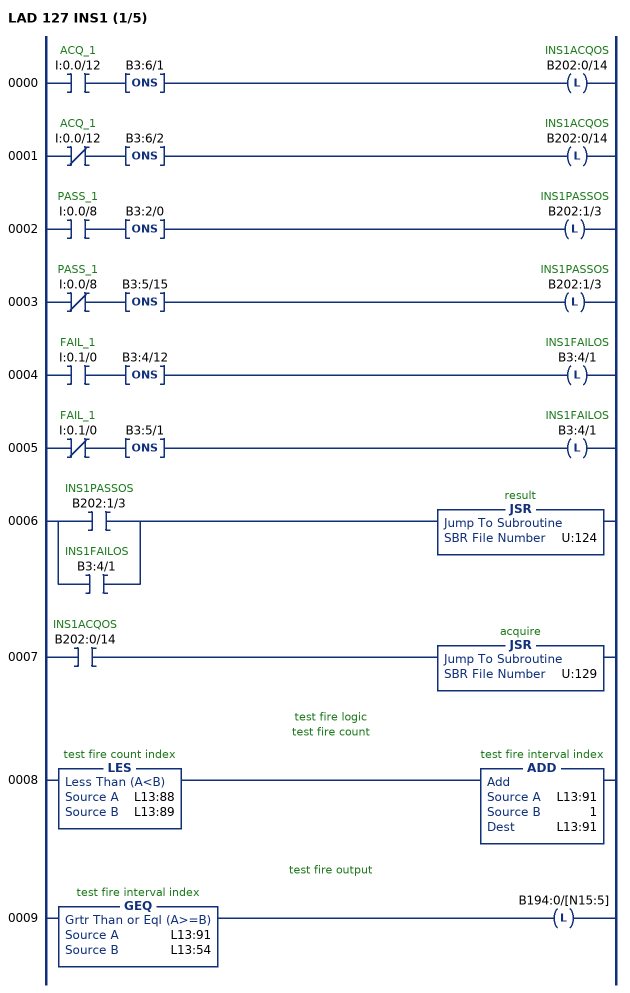
% Rung: 0 %
SOR XIC I:0.0/12 ONS B3:6/1 OTL B202:0/14 EOR
%   I:0.0/12  ACQ_1 %
%   B202:0/14  INS1ACQOS %
% Rung: 1 %
SOR XIO I:0.0/12 ONS B3:6/2 OTL B202:0/14 EOR
%   I:0.0/12  ACQ_1 %
%   B202:0/14  INS1ACQOS %
% Rung: 2 %
SOR XIC I:0.0/8 ONS B3:2/0 OTL B202:1/3 EOR
%   I:0.0/8  PASS_1 %
%   B202:1/3  INS1PASSOS %
% Rung: 3 %
SOR XIO I:0.0/8 ONS B3:5/15 OTL B202:1/3 EOR
%   I:0.0/8  PASS_1 %
%   B202:1/3  INS1PASSOS %
% Rung: 4 %
SOR XIC I:0.1/0 ONS B3:4/12 OTL B3:4/1 EOR
%   I:0.1/0  FAIL_1 %
%   B3:4/1  INS1FAILOS %
% Rung: 5 %
SOR XIO I:0.1/0 ONS B3:5/1 OTL B3:4/1 EOR
%   I:0.1/0  FAIL_1 %
%   B3:4/1  INS1FAILOS %
% Rung: 6 %
SOR BST XIC B202:1/3 NXB XIC B3:4/1 BND JSR U:124 EOR
%   B202:1/3  INS1PASSOS %
%   B3:4/1  INS1FAILOS %
%   U:124  "result" %
% Rung: 7 %
SOR XIC B202:0/14 JSR U:129 EOR
%   B202:0/14  INS1ACQOS %
%   U:129  "acquire" %
% Rung: 8 %
% test fire logic
% 
% test fire count %
SOR LES L13:88 L13:89 ADD L13:91 1 L13:91 EOR
%   L13:88  "test fire count index" %
%   L13:89  "test fire count" %
%   L13:91  "test fire interval index" %
% Rung: 9 %
% test fire output %
SOR GEQ L13:91 L13:54 OTL B194:0/[N15:5] EOR
%   L13:91  "test fire interval index" %
%   L13:54  "test fire interval" %
%   N15:5  INS_1_TRIG_LOC %

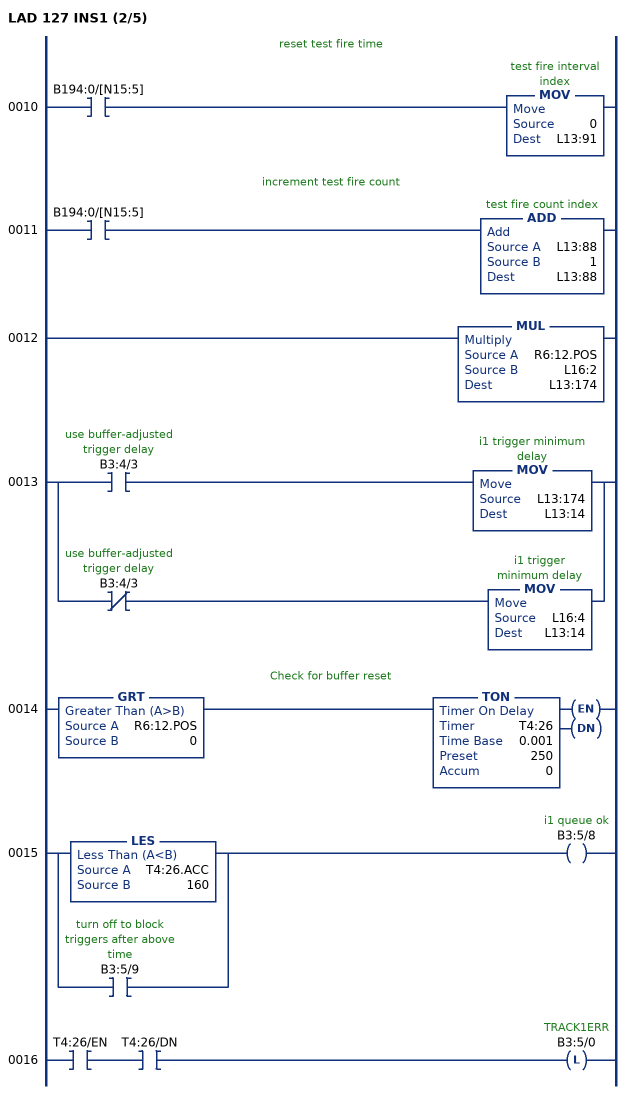
% Rung: 10 %
% reset test fire time %
SOR XIC B194:0/[N15:5] MOV 0 L13:91 EOR
%   N15:5  INS_1_TRIG_LOC %
%   L13:91  "test fire interval index" %
% Rung: 11 %
% increment test fire count %
SOR XIC B194:0/[N15:5] ADD L13:88 1 L13:88 EOR
%   N15:5  INS_1_TRIG_LOC %
%   L13:88  "test fire count index" %
% Rung: 12 %
SOR MUL R6:12.POS L16:2 L13:174 EOR
%   L16:2  TRIG_DELAY_Q_MULTI %
% Rung: 13 %
SOR BST XIC B3:4/3 MOV L13:174 L13:14 NXB XIO B3:4/3 MOV L16:4 L13:14 BND EOR
%   B3:4/3  "use buffer-adjusted trigger delay" %
%   L13:14  "i1 trigger minimum delay" %
%   L16:4  TRIG_DELAY_FLAT_RATE %
% Rung: 14 %
% Check for buffer reset %
SOR GRT R6:12.POS 0 TON T4:26 0.001 250 0 EOR
% Rung: 15 %
SOR BST LES T4:26.ACC 160 NXB XIC B3:5/9 BND OTE B3:5/8 EOR
%   B3:5/9  "turn off to block triggers after above time" %
%   B3:5/8  "i1 queue ok" %
% Rung: 16 %
SOR XIC T4:26/EN XIC T4:26/DN OTL B3:5/0 EOR
%   B3:5/0  TRACK1ERR %

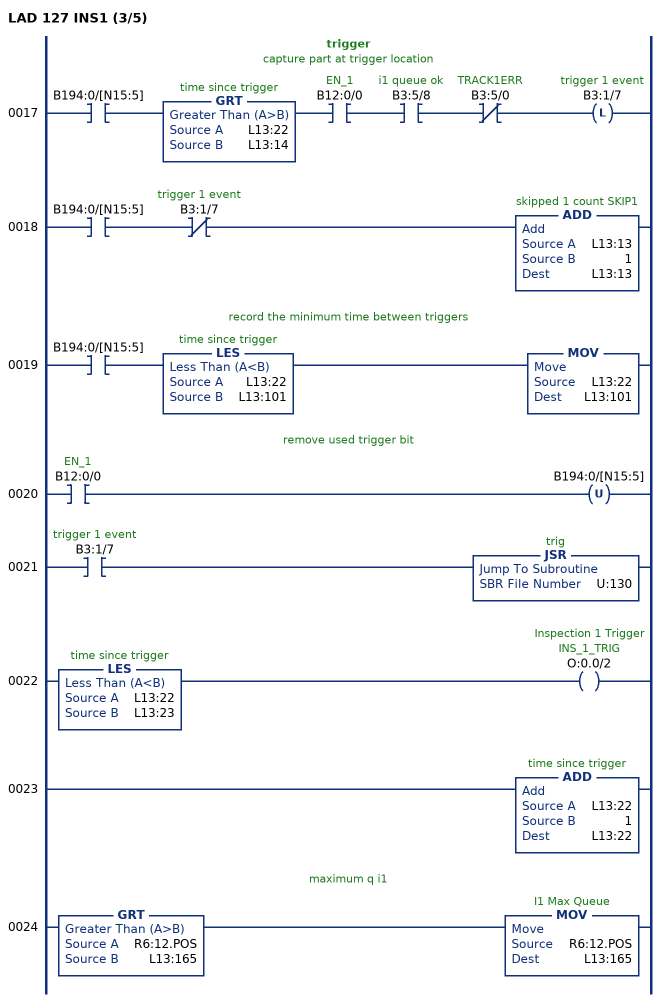
% Rung: 17 %
% TITLE: trigger %
% capture part at trigger location %
SOR XIC B194:0/[N15:5] GRT L13:22 L13:14 XIC B12:0/0 XIC B3:5/8 XIO B3:5/0 OTL B3:1/7 EOR
%   N15:5  INS_1_TRIG_LOC %
%   L13:22  "time since trigger" %
%   L13:14  "i1 trigger minimum delay" %
%   B12:0/0  EN_1 %
%   B3:5/8  "i1 queue ok" %
%   B3:5/0  TRACK1ERR %
%   B3:1/7  "trigger 1 event" %
% Rung: 18 %
SOR XIC B194:0/[N15:5] XIO B3:1/7 ADD L13:13 1 L13:13 EOR
%   N15:5  INS_1_TRIG_LOC %
%   B3:1/7  "trigger 1 event" %
%   L13:13  SKIP1  "skipped 1 count" %
% Rung: 19 %
% record the minimum time between triggers %
SOR XIC B194:0/[N15:5] LES L13:22 L13:101 MOV L13:22 L13:101 EOR
%   N15:5  INS_1_TRIG_LOC %
%   L13:22  "time since trigger" %
% Rung: 20 %
% remove used trigger bit %
SOR XIC B12:0/0 OTU B194:0/[N15:5] EOR
%   B12:0/0  EN_1 %
%   N15:5  INS_1_TRIG_LOC %
% Rung: 21 %
SOR XIC B3:1/7 JSR U:130 EOR
%   B3:1/7  "trigger 1 event" %
%   U:130  "trig" %
% Rung: 22 %
SOR LES L13:22 L13:23 OTE O:0.0/2 EOR
%   L13:22  "time since trigger" %
%   L13:23  "trigger on time" %
%   O:0.0/2  INS_1_TRIG  "Inspection 1 Trigger" %
% Rung: 23 %
SOR ADD L13:22 1 L13:22 EOR
%   L13:22  "time since trigger" %
% Rung: 24 %
% maximum q i1 %
SOR GRT R6:12.POS L13:165 MOV R6:12.POS L13:165 EOR
%   L13:165  "I1 Max Queue" %

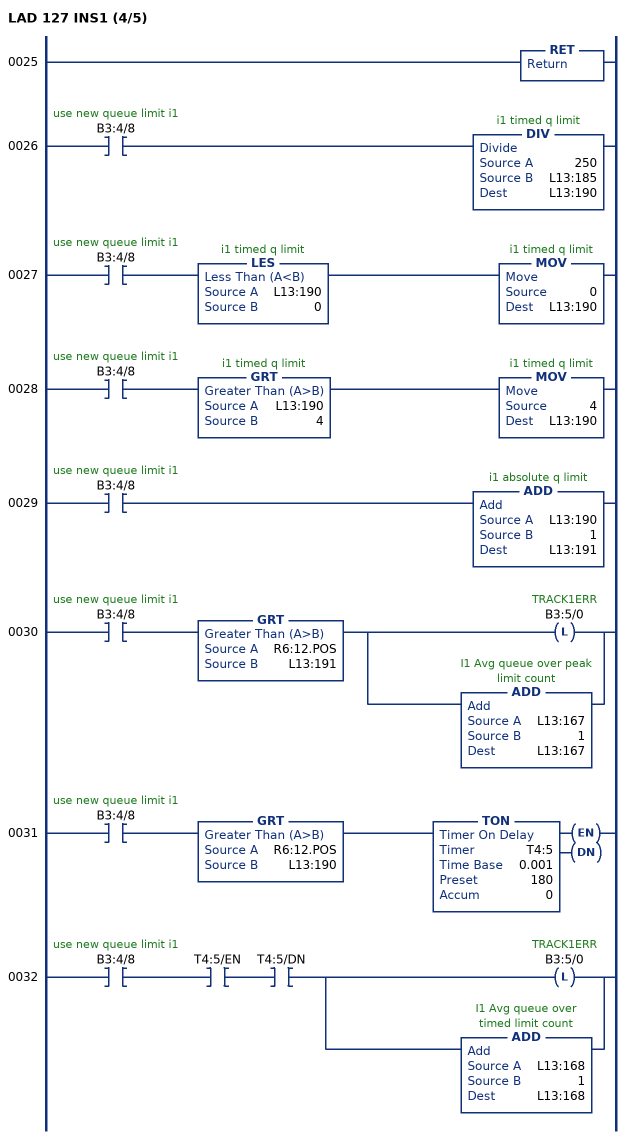
% Rung: 25 %
SOR RET EOR
% Rung: 26 %
SOR XIC B3:4/8 DIV 250 L13:185 L13:190 EOR
%   B3:4/8  "use new queue limit i1" %
%   L13:185  I1_TBT  "i1 average time between triggers" %
%   L13:190  "i1 timed q limit" %
% Rung: 27 %
SOR XIC B3:4/8 LES L13:190 0 MOV 0 L13:190 EOR
%   B3:4/8  "use new queue limit i1" %
%   L13:190  "i1 timed q limit" %
% Rung: 28 %
SOR XIC B3:4/8 GRT L13:190 4 MOV 4 L13:190 EOR
%   B3:4/8  "use new queue limit i1" %
%   L13:190  "i1 timed q limit" %
% Rung: 29 %
SOR XIC B3:4/8 ADD L13:190 1 L13:191 EOR
%   B3:4/8  "use new queue limit i1" %
%   L13:190  "i1 timed q limit" %
%   L13:191  "i1 absolute q limit" %
% Rung: 30 %
SOR XIC B3:4/8 GRT R6:12.POS L13:191 BST OTL B3:5/0 NXB ADD L13:167 1 L13:167 BND EOR
%   B3:4/8  "use new queue limit i1" %
%   L13:191  "i1 absolute q limit" %
%   B3:5/0  TRACK1ERR %
%   L13:167  "I1 Avg queue over peak limit count" %
% Rung: 31 %
SOR XIC B3:4/8 GRT R6:12.POS L13:190 TON T4:5 0.001 180 0 EOR
%   B3:4/8  "use new queue limit i1" %
%   L13:190  "i1 timed q limit" %
% Rung: 32 %
SOR XIC B3:4/8 XIC T4:5/EN XIC T4:5/DN BST OTL B3:5/0 NXB ADD L13:168 1 L13:168 BND EOR
%   B3:4/8  "use new queue limit i1" %
%   B3:5/0  TRACK1ERR %
%   L13:168  "I1 Avg queue over timed limit count" %

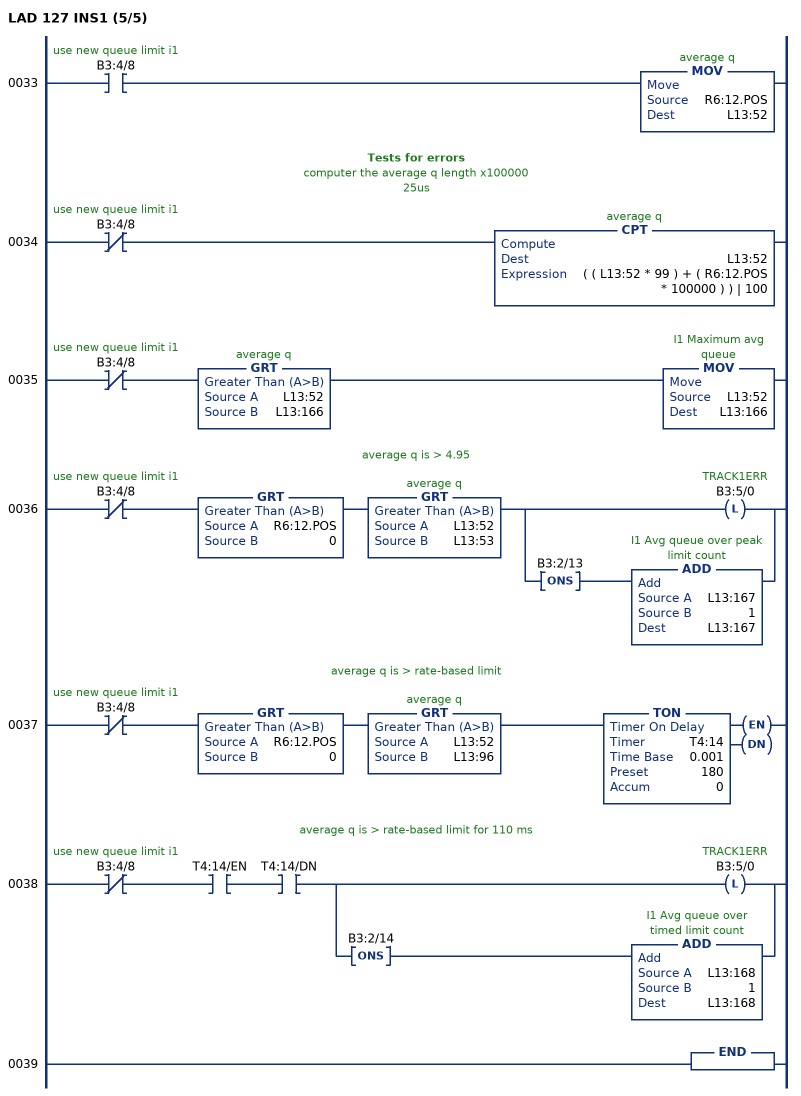
% Rung: 33 %
SOR XIC B3:4/8 MOV R6:12.POS L13:52 EOR
%   B3:4/8  "use new queue limit i1" %
%   L13:52  "average q" %
% Rung: 34 %
% TITLE: Tests for errors %
% computer the average q length x100000
% 25us %
SOR XIO B3:4/8 CPT L13:52 " ( ( L13:52 * 99 ) + ( R6:12.POS * 100000 ) ) | 100 " EOR
%   B3:4/8  "use new queue limit i1" %
%   L13:52  "average q" %
% Rung: 35 %
SOR XIO B3:4/8 GRT L13:52 L13:166 MOV L13:52 L13:166 EOR
%   B3:4/8  "use new queue limit i1" %
%   L13:52  "average q" %
%   L13:166  "I1 Maximum avg queue" %
% Rung: 36 %
% average q is > 4.95 %
SOR XIO B3:4/8 GRT R6:12.POS 0 GRT L13:52 L13:53 BST OTL B3:5/0 NXB ONS B3:2/13 ADD L13:167 1 L13:167 BND EOR
%   B3:4/8  "use new queue limit i1" %
%   L13:52  "average q" %
%   B3:5/0  TRACK1ERR %
%   L13:167  "I1 Avg queue over peak limit count" %
% Rung: 37 %
% average q is > rate-based limit %
SOR XIO B3:4/8 GRT R6:12.POS 0 GRT L13:52 L13:96 TON T4:14 0.001 180 0 EOR
%   B3:4/8  "use new queue limit i1" %
%   L13:52  "average q" %
%   L13:96  "i1 timed queue limit" %
% Rung: 38 %
% average q is > rate-based limit for 110 ms %
SOR XIO B3:4/8 XIC T4:14/EN XIC T4:14/DN BST OTL B3:5/0 NXB ONS B3:2/14 ADD L13:168 1 L13:168 BND EOR
%   B3:4/8  "use new queue limit i1" %
%   B3:5/0  TRACK1ERR %
%   L13:168  "I1 Avg queue over timed limit count" %
% Rung: 39 %
SOR END EOR

LADDER 128 "INS1PASS"
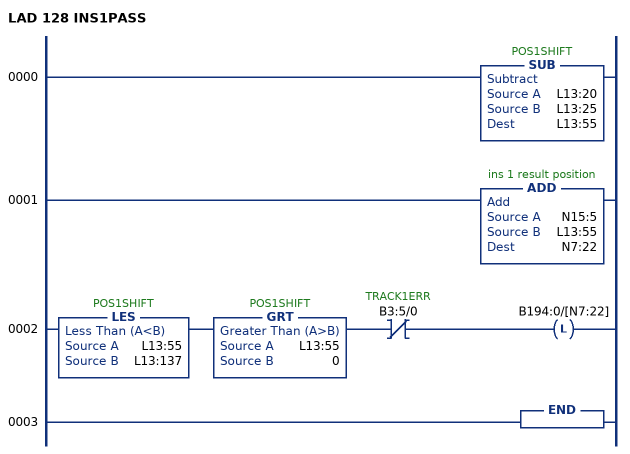
% Rung: 0 %
SOR SUB L13:20 L13:25 L13:55 EOR
%   L13:20  BOT_POSITION %
%   L13:25  POS1  "last acquisition position stamp" %
%   L13:55  POS1SHIFT %
% Rung: 1 %
SOR ADD N15:5 L13:55 N7:22 EOR
%   N15:5  INS_1_TRIG_LOC %
%   L13:55  POS1SHIFT %
%   N7:22  "ins 1 result position" %
% Rung: 2 %
SOR LES L13:55 L13:137 GRT L13:55 0 XIO B3:5/0 OTL B194:0/[N7:22] EOR
%   L13:55  POS1SHIFT %
%   B3:5/0  TRACK1ERR %
%   N7:22  "ins 1 result position" %
% Rung: 3 %
SOR END EOR

LADDER 129 "INS1ACQ"
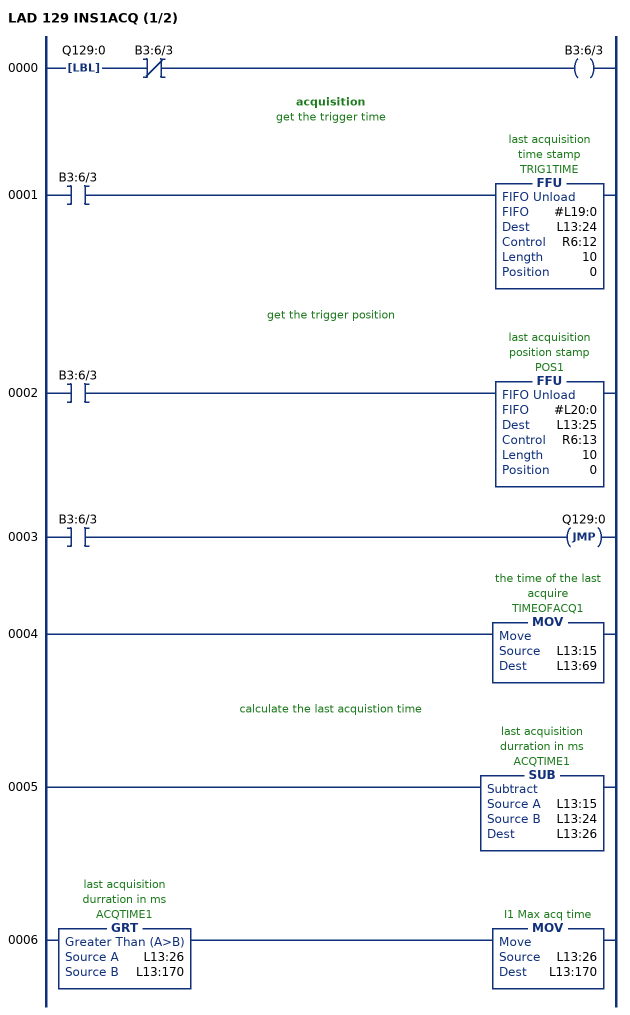
% Rung: 0 %
SOR LBL Q129:0 XIO B3:6/3 OTE B3:6/3 EOR
% Rung: 1 %
% TITLE: acquisition %
% get the trigger time %
SOR XIC B3:6/3 FFU #L19:0 L13:24 R6:12 10 0 EOR
%   L13:24  TRIG1TIME  "last acquisition time stamp" %
% Rung: 2 %
% get the trigger position %
SOR XIC B3:6/3 FFU #L20:0 L13:25 R6:13 10 0 EOR
%   L13:25  POS1  "last acquisition position stamp" %
% Rung: 3 %
SOR XIC B3:6/3 JMP Q129:0 EOR
% Rung: 4 %
SOR MOV L13:15 L13:69 EOR
%   L13:15  THE_TIME %
%   L13:69  TIMEOFACQ1  "the time of the last acquire" %
% Rung: 5 %
% calculate the last acquistion time %
SOR SUB L13:15 L13:24 L13:26 EOR
%   L13:15  THE_TIME %
%   L13:24  TRIG1TIME  "last acquisition time stamp" %
%   L13:26  ACQTIME1  "last acquisition durration in ms" %
% Rung: 6 %
SOR GRT L13:26 L13:170 MOV L13:26 L13:170 EOR
%   L13:26  ACQTIME1  "last acquisition durration in ms" %
%   L13:170  "I1 Max acq time" %

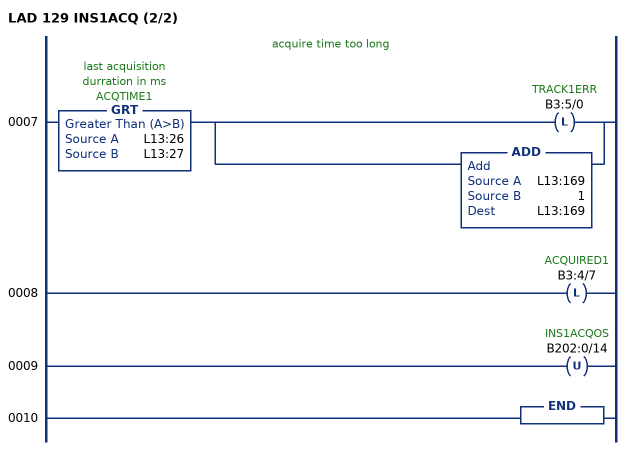
% Rung: 7 %
% acquire time too long %
SOR GRT L13:26 L13:27 BST OTL B3:5/0 NXB ADD L13:169 1 L13:169 BND EOR
%   L13:26  ACQTIME1  "last acquisition durration in ms" %
%   L13:27  "max acquisition time in ms" %
%   B3:5/0  TRACK1ERR %
% Rung: 8 %
SOR OTL B3:4/7 EOR
%   B3:4/7  ACQUIRED1 %
% Rung: 9 %
SOR OTU B202:0/14 EOR
%   B202:0/14  INS1ACQOS %
% Rung: 10 %
SOR END EOR

LADDER 130 "INS1TRIG"
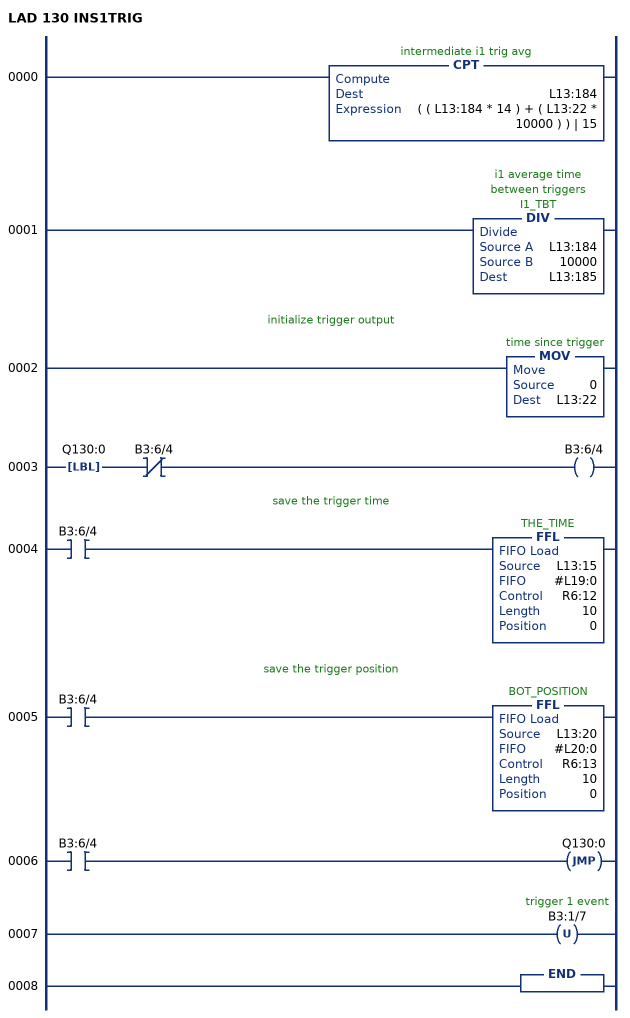
% Rung: 0 %
SOR CPT L13:184 " ( ( L13:184 * 14 ) + ( L13:22 * 10000 ) ) | 15 " EOR
%   L13:184  "intermediate i1 trig avg" %
%   L13:22  "time since trigger" %
% Rung: 1 %
SOR DIV L13:184 10000 L13:185 EOR
%   L13:184  "intermediate i1 trig avg" %
%   L13:185  I1_TBT  "i1 average time between triggers" %
% Rung: 2 %
% initialize trigger output %
SOR MOV 0 L13:22 EOR
%   L13:22  "time since trigger" %
% Rung: 3 %
SOR LBL Q130:0 XIO B3:6/4 OTE B3:6/4 EOR
% Rung: 4 %
% save the trigger time %
SOR XIC B3:6/4 FFL L13:15 #L19:0 R6:12 10 0 EOR
%   L13:15  THE_TIME %
% Rung: 5 %
% save the trigger position %
SOR XIC B3:6/4 FFL L13:20 #L20:0 R6:13 10 0 EOR
%   L13:20  BOT_POSITION %
% Rung: 6 %
SOR XIC B3:6/4 JMP Q130:0 EOR
% Rung: 7 %
SOR OTU B3:1/7 EOR
%   B3:1/7  "trigger 1 event" %
% Rung: 8 %
SOR END EOR

LADDER 131 "XFER"
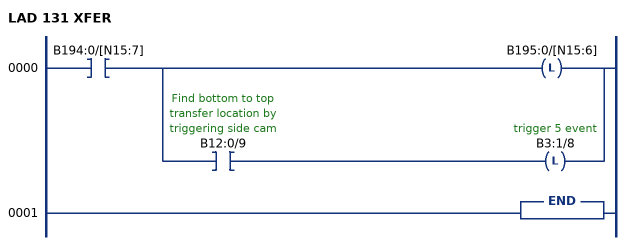
% Rung: 0 %
SOR XIC B194:0/[N15:7] BST OTL B195:0/[N15:6] NXB XIC B12:0/9 OTL B3:1/8 BND EOR
%   N15:7  XFER_OUT_LOC %
%   N15:6  XFER_IN_LOC %
%   B12:0/9  "Find bottom to top transfer location by triggering side cam" %
%   B3:1/8  "trigger 5 event" %
% Rung: 1 %
SOR END EOR

LADDER 140 "TOPOPTIC"
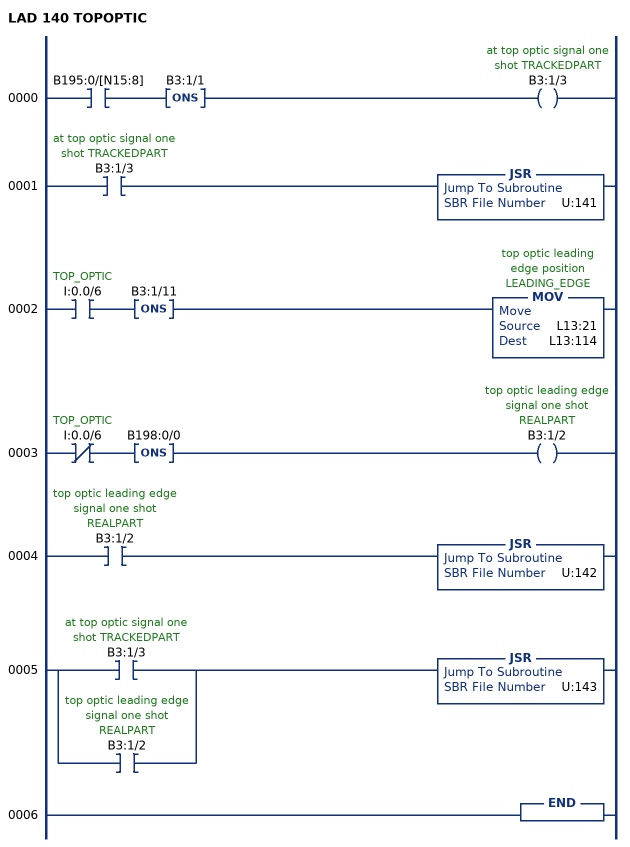
% Rung: 0 %
SOR XIC B195:0/[N15:8] ONS B3:1/1 OTE B3:1/3 EOR
%   N15:8  TOP_OPTIC_LOC %
%   B3:1/3  TRACKEDPART  "at top optic signal one shot" %
% Rung: 1 %
SOR XIC B3:1/3 JSR U:141 EOR
%   B3:1/3  TRACKEDPART  "at top optic signal one shot" %
% Rung: 2 %
SOR XIC I:0.0/6 ONS B3:1/11 MOV L13:21 L13:114 EOR
%   I:0.0/6  TOP_OPTIC %
%   L13:21  TOP_POSITION %
%   L13:114  LEADING_EDGE  "top optic leading edge position" %
% Rung: 3 %
SOR XIO I:0.0/6 ONS B198:0/0 OTE B3:1/2 EOR
%   I:0.0/6  TOP_OPTIC %
%   B3:1/2  REALPART  "top optic leading edge signal one shot" %
% Rung: 4 %
SOR XIC B3:1/2 JSR U:142 EOR
%   B3:1/2  REALPART  "top optic leading edge signal one shot" %
% Rung: 5 %
SOR BST XIC B3:1/3 NXB XIC B3:1/2 BND JSR U:143 EOR
%   B3:1/3  TRACKEDPART  "at top optic signal one shot" %
%   B3:1/2  REALPART  "top optic leading edge signal one shot" %
% Rung: 6 %
SOR END EOR

LADDER 141 "TOPOPVERT"
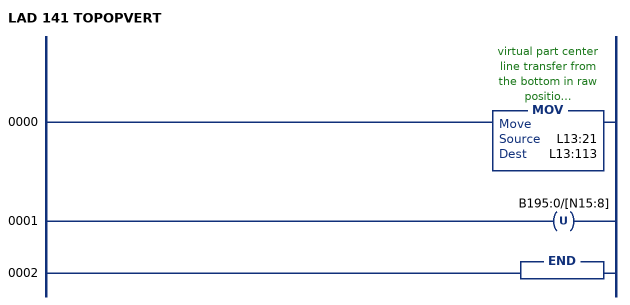
% Rung: 0 %
SOR MOV L13:21 L13:113 EOR
%   L13:21  TOP_POSITION %
%   L13:113  VERTUAL_PT_RAW_CL  "virtual part center line transfer from the bottom in raw position" %
% Rung: 1 %
SOR OTU B195:0/[N15:8] EOR
%   N15:8  TOP_OPTIC_LOC %
% Rung: 2 %
SOR END EOR

LADDER 142 "TOPOPREAL"
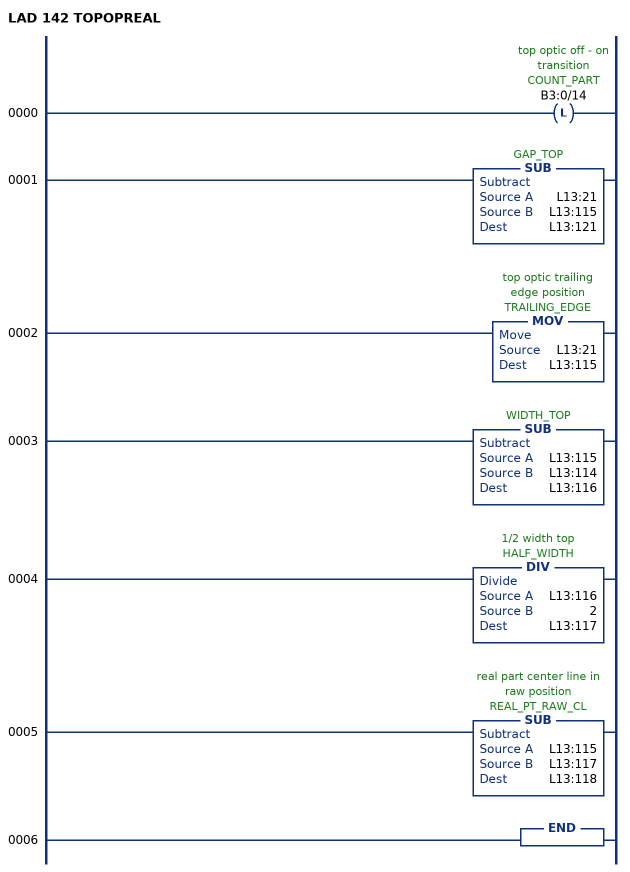
% Rung: 0 %
SOR OTL B3:0/14 EOR
%   B3:0/14  COUNT_PART  "top optic off - on transition" %
% Rung: 1 %
SOR SUB L13:21 L13:115 L13:121 EOR
%   L13:21  TOP_POSITION %
%   L13:115  TRAILING_EDGE  "top optic trailing edge position" %
%   L13:121  GAP_TOP %
% Rung: 2 %
SOR MOV L13:21 L13:115 EOR
%   L13:21  TOP_POSITION %
%   L13:115  TRAILING_EDGE  "top optic trailing edge position" %
% Rung: 3 %
SOR SUB L13:115 L13:114 L13:116 EOR
%   L13:115  TRAILING_EDGE  "top optic trailing edge position" %
%   L13:114  LEADING_EDGE  "top optic leading edge position" %
%   L13:116  WIDTH_TOP %
% Rung: 4 %
SOR DIV L13:116 2 L13:117 EOR
%   L13:116  WIDTH_TOP %
%   L13:117  HALF_WIDTH  "1/2 width top" %
% Rung: 5 %
SOR SUB L13:115 L13:117 L13:118 EOR
%   L13:115  TRAILING_EDGE  "top optic trailing edge position" %
%   L13:117  HALF_WIDTH  "1/2 width top" %
%   L13:118  REAL_PT_RAW_CL  "real part center line in raw position" %
% Rung: 6 %
SOR END EOR

LADDER 143 "TOPOPTEST"
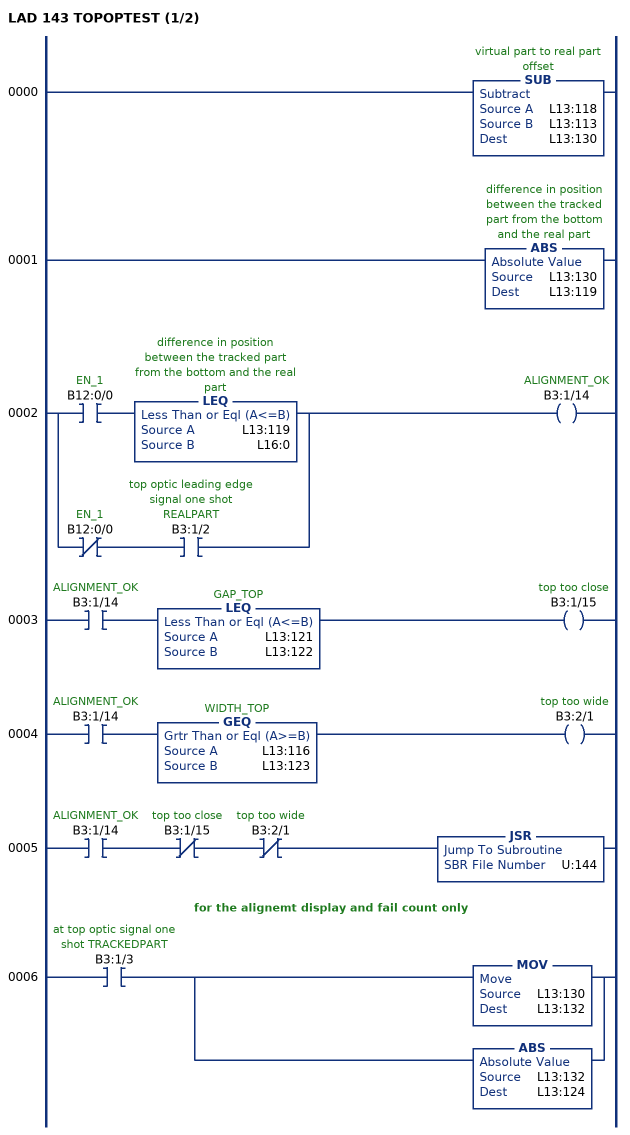
% Rung: 0 %
SOR SUB L13:118 L13:113 L13:130 EOR
%   L13:118  REAL_PT_RAW_CL  "real part center line in raw position" %
%   L13:113  VERTUAL_PT_RAW_CL  "virtual part center line transfer from the bottom in raw position" %
%   L13:130  "virtual part to real part offset" %
% Rung: 1 %
SOR ABS L13:130 L13:119 EOR
%   L13:130  "virtual part to real part offset" %
%   L13:119  "difference in position between the tracked part from the bottom and the real part" %
% Rung: 2 %
SOR BST XIC B12:0/0 LEQ L13:119 L16:0 NXB XIO B12:0/0 XIC B3:1/2 BND OTE B3:1/14 EOR
%   B12:0/0  EN_1 %
%   L13:119  "difference in position between the tracked part from the bottom and the real part" %
%   L16:0  MAX_OFFSET %
%   B3:1/2  REALPART  "top optic leading edge signal one shot" %
%   B3:1/14  ALIGNMENT_OK %
% Rung: 3 %
SOR XIC B3:1/14 LEQ L13:121 L13:122 OTE B3:1/15 EOR
%   B3:1/14  ALIGNMENT_OK %
%   L13:121  GAP_TOP %
%   L13:122  MIN_GAP_TOP %
%   B3:1/15  "top too close" %
% Rung: 4 %
SOR XIC B3:1/14 GEQ L13:116 L13:123 OTE B3:2/1 EOR
%   B3:1/14  ALIGNMENT_OK %
%   L13:116  WIDTH_TOP %
%   L13:123  MAX_WIDTH_TOP %
%   B3:2/1  "top too wide" %
% Rung: 5 %
SOR XIC B3:1/14 XIO B3:1/15 XIO B3:2/1 JSR U:144 EOR
%   B3:1/14  ALIGNMENT_OK %
%   B3:1/15  "top too close" %
%   B3:2/1  "top too wide" %
% Rung: 6 %
% TITLE: for the alignemt display and fail count only %
SOR XIC B3:1/3 BST MOV L13:130 L13:132 NXB ABS L13:132 L13:124 BND EOR
%   B3:1/3  TRACKEDPART  "at top optic signal one shot" %
%   L13:130  "virtual part to real part offset" %

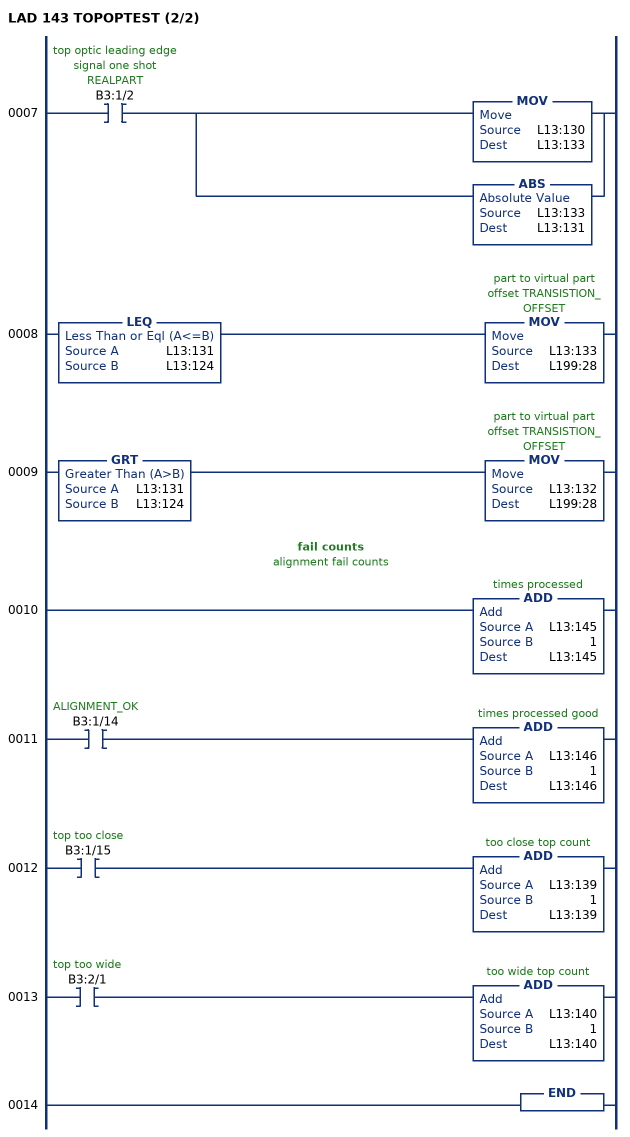
% Rung: 7 %
SOR XIC B3:1/2 BST MOV L13:130 L13:133 NXB ABS L13:133 L13:131 BND EOR
%   B3:1/2  REALPART  "top optic leading edge signal one shot" %
%   L13:130  "virtual part to real part offset" %
% Rung: 8 %
SOR LEQ L13:131 L13:124 MOV L13:133 L199:28 EOR
%   L199:28  TRANSISTION_OFFSET  "part to virtual part offset" %
% Rung: 9 %
SOR GRT L13:131 L13:124 MOV L13:132 L199:28 EOR
%   L199:28  TRANSISTION_OFFSET  "part to virtual part offset" %
% Rung: 10 %
% TITLE: fail counts %
% alignment fail counts %
SOR ADD L13:145 1 L13:145 EOR
%   L13:145  "times processed" %
% Rung: 11 %
SOR XIC B3:1/14 ADD L13:146 1 L13:146 EOR
%   B3:1/14  ALIGNMENT_OK %
%   L13:146  "times processed good" %
% Rung: 12 %
SOR XIC B3:1/15 ADD L13:139 1 L13:139 EOR
%   B3:1/15  "top too close" %
%   L13:139  "too close top count" %
% Rung: 13 %
SOR XIC B3:2/1 ADD L13:140 1 L13:140 EOR
%   B3:2/1  "top too wide" %
%   L13:140  "too wide top count" %
% Rung: 14 %
SOR END EOR

LADDER 144 "TOPOPOKAY"
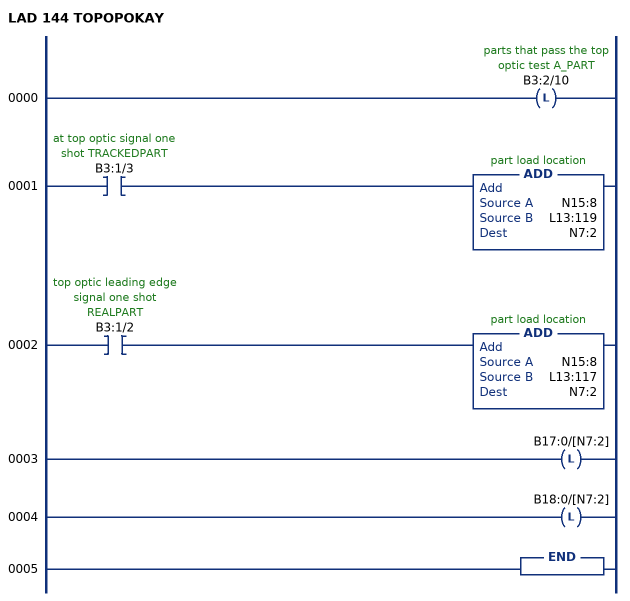
% Rung: 0 %
SOR OTL B3:2/10 EOR
%   B3:2/10  A_PART  "parts that pass the top optic test" %
% Rung: 1 %
SOR XIC B3:1/3 ADD N15:8 L13:119 N7:2 EOR
%   B3:1/3  TRACKEDPART  "at top optic signal one shot" %
%   N15:8  TOP_OPTIC_LOC %
%   L13:119  "difference in position between the tracked part from the bottom and the real part" %
%   N7:2  "part load location" %
% Rung: 2 %
SOR XIC B3:1/2 ADD N15:8 L13:117 N7:2 EOR
%   B3:1/2  REALPART  "top optic leading edge signal one shot" %
%   N15:8  TOP_OPTIC_LOC %
%   L13:117  HALF_WIDTH  "1/2 width top" %
%   N7:2  "part load location" %
% Rung: 3 %
SOR OTL B17:0/[N7:2] EOR
%   N7:2  "part load location" %
% Rung: 4 %
SOR OTL B18:0/[N7:2] EOR
%   N7:2  "part load location" %
% Rung: 5 %
SOR END EOR

LADDER 149 "INS5RESULT"
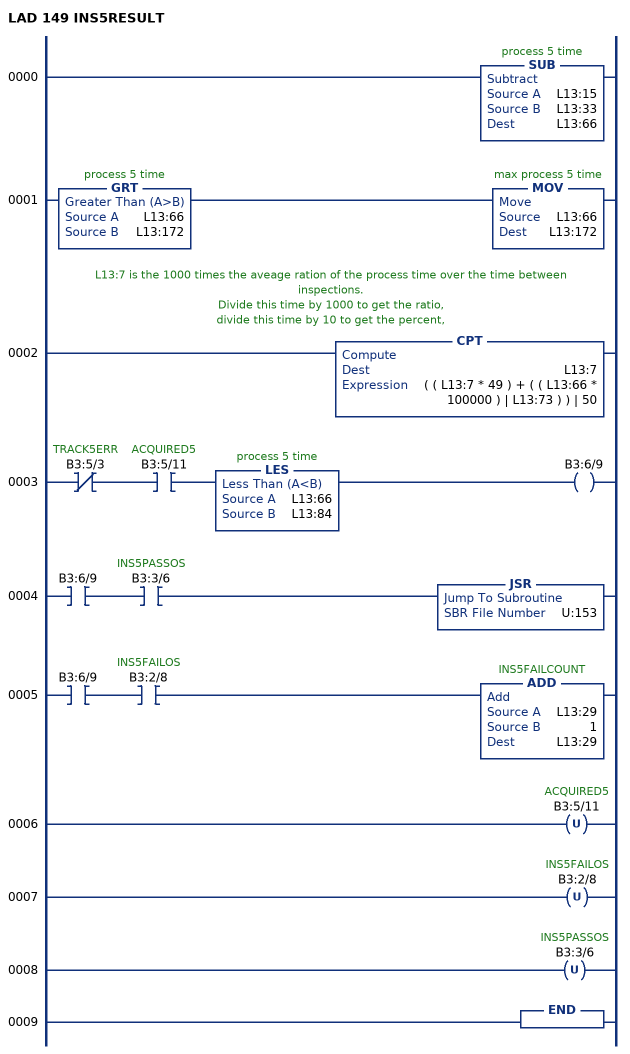
% Rung: 0 %
SOR SUB L13:15 L13:33 L13:66 EOR
%   L13:15  THE_TIME %
%   L13:33  TIMEOFACQ5  "the time of the last acquire" %
%   L13:66  "process 5 time" %
% Rung: 1 %
SOR GRT L13:66 L13:172 MOV L13:66 L13:172 EOR
%   L13:66  "process 5 time" %
%   L13:172  "max process 5 time" %
% Rung: 2 %
% L13:7 is the 1000 times the aveage ration of the process time over the time between inspections.
% Divide this time by 1000 to get the ratio,
% divide this time by 10 to get the percent, %
SOR CPT L13:7 " ( ( L13:7 * 49 ) + ( ( L13:66 * 100000 ) | L13:73 ) ) | 50 " EOR
%   L13:66  "process 5 time" %
%   L13:73  TBI  "the time between inspections in 0.000,01 seconds or 1/6000000 minutes." %
% Rung: 3 %
SOR XIO B3:5/3 XIC B3:5/11 LES L13:66 L13:84 OTE B3:6/9 EOR
%   B3:5/3  TRACK5ERR %
%   B3:5/11  ACQUIRED5 %
%   L13:66  "process 5 time" %
% Rung: 4 %
SOR XIC B3:6/9 XIC B3:3/6 JSR U:153 EOR
%   B3:3/6  INS5PASSOS %
% Rung: 5 %
SOR XIC B3:6/9 XIC B3:2/8 ADD L13:29 1 L13:29 EOR
%   B3:2/8  INS5FAILOS %
%   L13:29  INS5FAILCOUNT %
% Rung: 6 %
SOR OTU B3:5/11 EOR
%   B3:5/11  ACQUIRED5 %
% Rung: 7 %
SOR OTU B3:2/8 EOR
%   B3:2/8  INS5FAILOS %
% Rung: 8 %
SOR OTU B3:3/6 EOR
%   B3:3/6  INS5PASSOS %
% Rung: 9 %
SOR END EOR

LADDER 150 "FIXERR5"
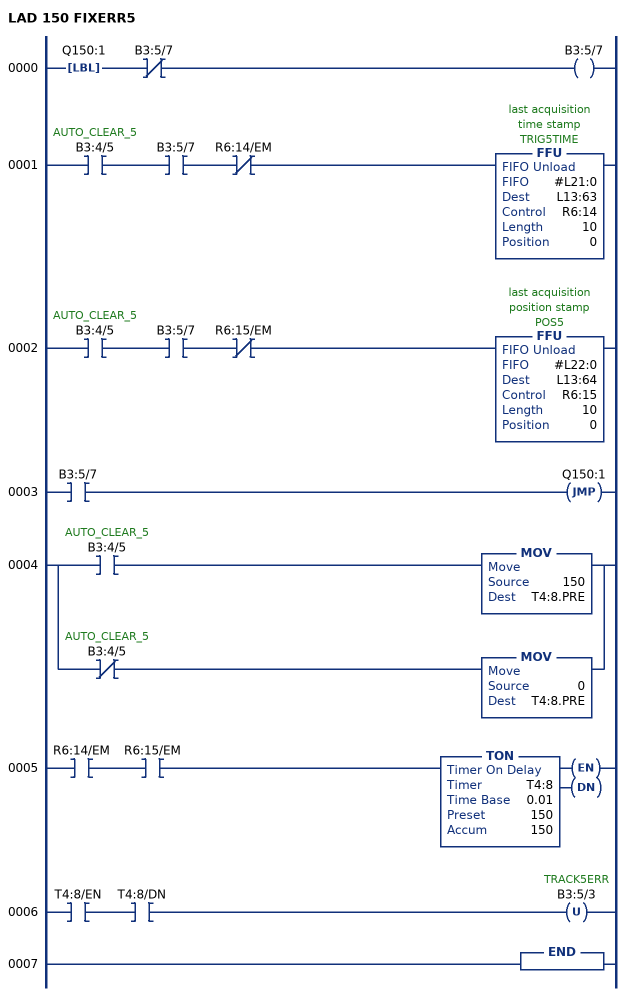
% Rung: 0 %
SOR LBL Q150:1 XIO B3:5/7 OTE B3:5/7 EOR
% Rung: 1 %
SOR XIC B3:4/5 XIC B3:5/7 XIO R6:14/EM FFU #L21:0 L13:63 R6:14 10 0 EOR
%   B3:4/5  AUTO_CLEAR_5 %
%   L13:63  TRIG5TIME  "last acquisition time stamp" %
% Rung: 2 %
SOR XIC B3:4/5 XIC B3:5/7 XIO R6:15/EM FFU #L22:0 L13:64 R6:15 10 0 EOR
%   B3:4/5  AUTO_CLEAR_5 %
%   L13:64  POS5  "last acquisition position stamp" %
% Rung: 3 %
SOR XIC B3:5/7 JMP Q150:1 EOR
% Rung: 4 %
SOR BST XIC B3:4/5 MOV 150 T4:8.PRE NXB XIO B3:4/5 MOV 0 T4:8.PRE BND EOR
%   B3:4/5  AUTO_CLEAR_5 %
% Rung: 5 %
SOR XIC R6:14/EM XIC R6:15/EM TON T4:8 0.01 150 150 EOR
% Rung: 6 %
SOR XIC T4:8/EN XIC T4:8/DN OTU B3:5/3 EOR
%   B3:5/3  TRACK5ERR %
% Rung: 7 %
SOR END EOR

LADDER 152 "INS5"
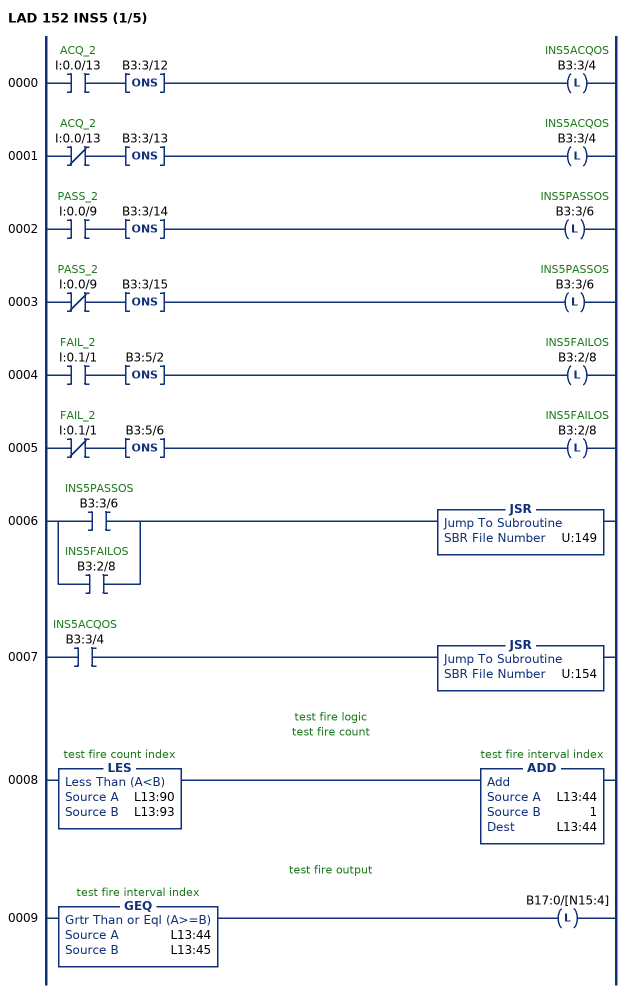
% Rung: 0 %
SOR XIC I:0.0/13 ONS B3:3/12 OTL B3:3/4 EOR
%   I:0.0/13  ACQ_2 %
%   B3:3/4  INS5ACQOS %
% Rung: 1 %
SOR XIO I:0.0/13 ONS B3:3/13 OTL B3:3/4 EOR
%   I:0.0/13  ACQ_2 %
%   B3:3/4  INS5ACQOS %
% Rung: 2 %
SOR XIC I:0.0/9 ONS B3:3/14 OTL B3:3/6 EOR
%   I:0.0/9  PASS_2 %
%   B3:3/6  INS5PASSOS %
% Rung: 3 %
SOR XIO I:0.0/9 ONS B3:3/15 OTL B3:3/6 EOR
%   I:0.0/9  PASS_2 %
%   B3:3/6  INS5PASSOS %
% Rung: 4 %
SOR XIC I:0.1/1 ONS B3:5/2 OTL B3:2/8 EOR
%   I:0.1/1  FAIL_2 %
%   B3:2/8  INS5FAILOS %
% Rung: 5 %
SOR XIO I:0.1/1 ONS B3:5/6 OTL B3:2/8 EOR
%   I:0.1/1  FAIL_2 %
%   B3:2/8  INS5FAILOS %
% Rung: 6 %
SOR BST XIC B3:3/6 NXB XIC B3:2/8 BND JSR U:149 EOR
%   B3:3/6  INS5PASSOS %
%   B3:2/8  INS5FAILOS %
% Rung: 7 %
SOR XIC B3:3/4 JSR U:154 EOR
%   B3:3/4  INS5ACQOS %
% Rung: 8 %
% test fire logic
% 
% test fire count %
SOR LES L13:90 L13:93 ADD L13:44 1 L13:44 EOR
%   L13:90  "test fire count index" %
%   L13:93  "test fire count" %
%   L13:44  "test fire interval index" %
% Rung: 9 %
% test fire output %
SOR GEQ L13:44 L13:45 OTL B17:0/[N15:4] EOR
%   L13:44  "test fire interval index" %
%   L13:45  "test fire interval" %
%   N15:4  INS_5_TRIG_LOC %

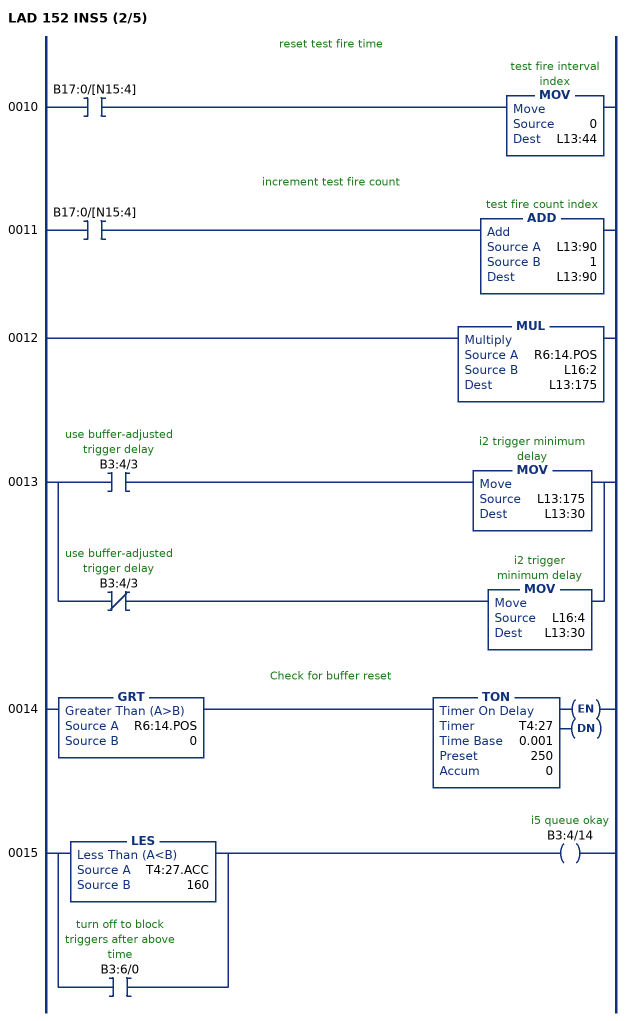
% Rung: 10 %
% reset test fire time %
SOR XIC B17:0/[N15:4] MOV 0 L13:44 EOR
%   N15:4  INS_5_TRIG_LOC %
%   L13:44  "test fire interval index" %
% Rung: 11 %
% increment test fire count %
SOR XIC B17:0/[N15:4] ADD L13:90 1 L13:90 EOR
%   N15:4  INS_5_TRIG_LOC %
%   L13:90  "test fire count index" %
% Rung: 12 %
SOR MUL R6:14.POS L16:2 L13:175 EOR
%   L16:2  TRIG_DELAY_Q_MULTI %
% Rung: 13 %
SOR BST XIC B3:4/3 MOV L13:175 L13:30 NXB XIO B3:4/3 MOV L16:4 L13:30 BND EOR
%   B3:4/3  "use buffer-adjusted trigger delay" %
%   L13:30  "i2 trigger minimum delay" %
%   L16:4  TRIG_DELAY_FLAT_RATE %
% Rung: 14 %
% Check for buffer reset %
SOR GRT R6:14.POS 0 TON T4:27 0.001 250 0 EOR
% Rung: 15 %
SOR BST LES T4:27.ACC 160 NXB XIC B3:6/0 BND OTE B3:4/14 EOR
%   B3:6/0  "turn off to block triggers after above time" %
%   B3:4/14  "i5 queue okay" %

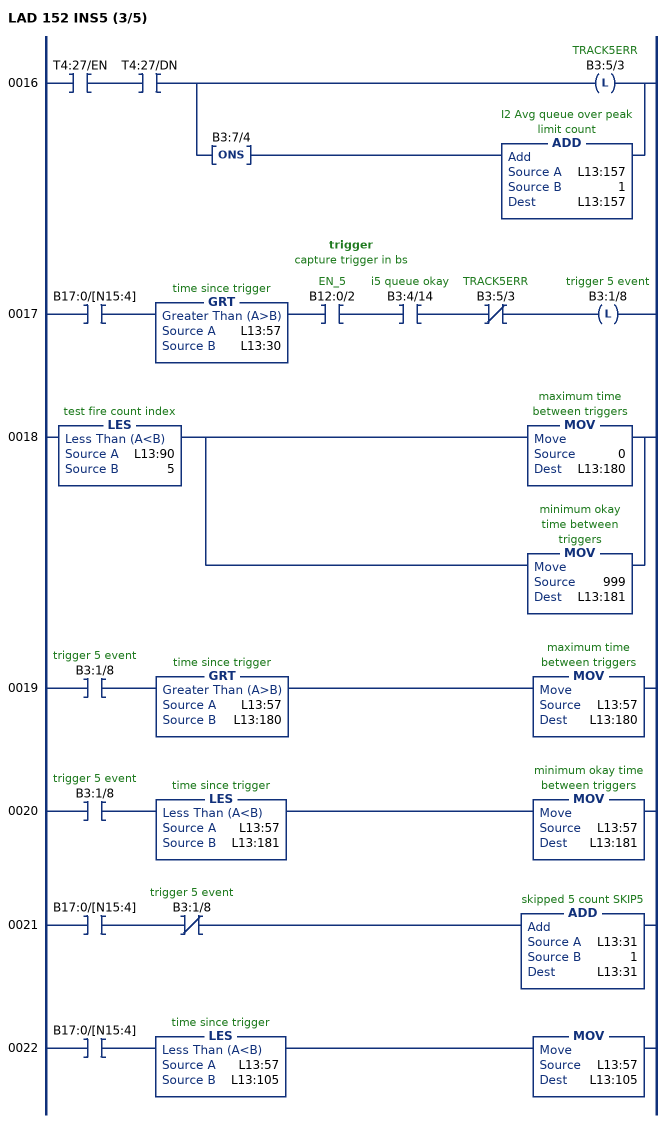
% Rung: 16 %
SOR XIC T4:27/EN XIC T4:27/DN BST OTL B3:5/3 NXB ONS B3:7/4 ADD L13:157 1 L13:157 BND EOR
%   B3:5/3  TRACK5ERR %
%   L13:157  "I2 Avg queue over peak limit count" %
% Rung: 17 %
% TITLE: trigger %
% capture trigger in bs %
SOR XIC B17:0/[N15:4] GRT L13:57 L13:30 XIC B12:0/2 XIC B3:4/14 XIO B3:5/3 OTL B3:1/8 EOR
%   N15:4  INS_5_TRIG_LOC %
%   L13:57  "time since trigger" %
%   L13:30  "i2 trigger minimum delay" %
%   B12:0/2  EN_5 %
%   B3:4/14  "i5 queue okay" %
%   B3:5/3  TRACK5ERR %
%   B3:1/8  "trigger 5 event" %
% Rung: 18 %
SOR LES L13:90 5 BST MOV 0 L13:180 NXB MOV 999 L13:181 BND EOR
%   L13:90  "test fire count index" %
%   L13:180  "maximum time between triggers" %
%   L13:181  "minimum okay time between triggers" %
% Rung: 19 %
SOR XIC B3:1/8 GRT L13:57 L13:180 MOV L13:57 L13:180 EOR
%   B3:1/8  "trigger 5 event" %
%   L13:57  "time since trigger" %
%   L13:180  "maximum time between triggers" %
% Rung: 20 %
SOR XIC B3:1/8 LES L13:57 L13:181 MOV L13:57 L13:181 EOR
%   B3:1/8  "trigger 5 event" %
%   L13:57  "time since trigger" %
%   L13:181  "minimum okay time between triggers" %
% Rung: 21 %
SOR XIC B17:0/[N15:4] XIO B3:1/8 ADD L13:31 1 L13:31 EOR
%   N15:4  INS_5_TRIG_LOC %
%   B3:1/8  "trigger 5 event" %
%   L13:31  SKIP5  "skipped 5 count" %
% Rung: 22 %
SOR XIC B17:0/[N15:4] LES L13:57 L13:105 MOV L13:57 L13:105 EOR
%   N15:4  INS_5_TRIG_LOC %
%   L13:57  "time since trigger" %

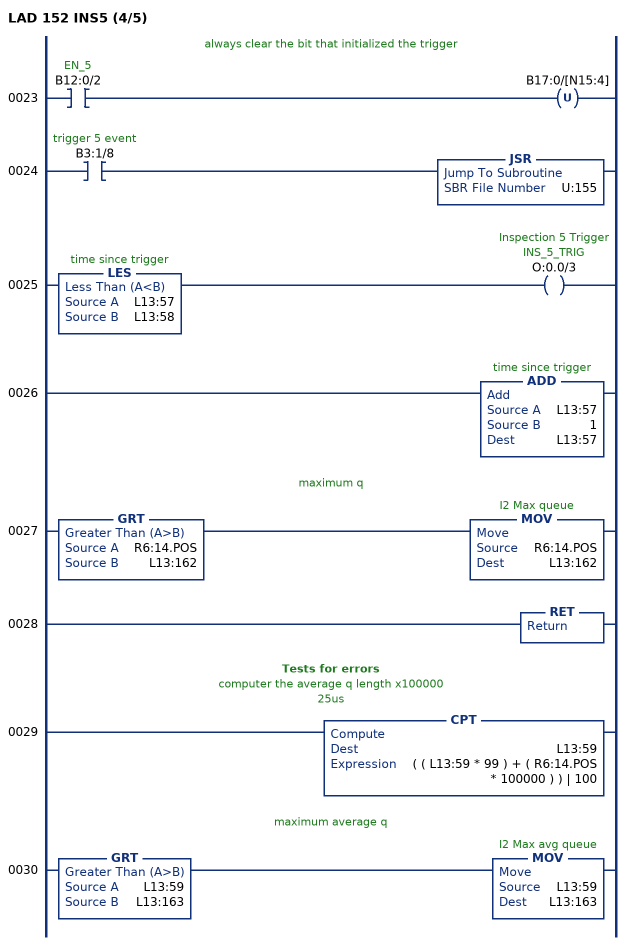
% Rung: 23 %
% always clear the bit that initialized the trigger %
SOR XIC B12:0/2 OTU B17:0/[N15:4] EOR
%   B12:0/2  EN_5 %
%   N15:4  INS_5_TRIG_LOC %
% Rung: 24 %
SOR XIC B3:1/8 JSR U:155 EOR
%   B3:1/8  "trigger 5 event" %
% Rung: 25 %
SOR LES L13:57 L13:58 OTE O:0.0/3 EOR
%   L13:57  "time since trigger" %
%   O:0.0/3  INS_5_TRIG  "Inspection 5 Trigger" %
% Rung: 26 %
SOR ADD L13:57 1 L13:57 EOR
%   L13:57  "time since trigger" %
% Rung: 27 %
% maximum q %
SOR GRT R6:14.POS L13:162 MOV R6:14.POS L13:162 EOR
%   L13:162  "I2 Max queue" %
% Rung: 28 %
SOR RET EOR
% Rung: 29 %
% TITLE: Tests for errors %
% computer the average q length x100000
% 25us %
SOR CPT L13:59 " ( ( L13:59 * 99 ) + ( R6:14.POS * 100000 ) ) | 100 " EOR
% Rung: 30 %
% maximum average q %
SOR GRT L13:59 L13:163 MOV L13:59 L13:163 EOR
%   L13:163  "I2 Max avg queue" %

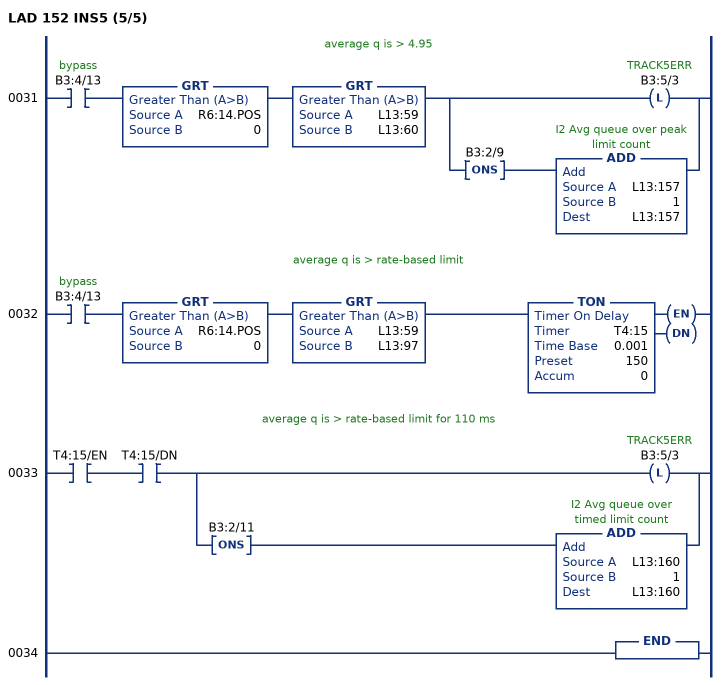
% Rung: 31 %
% average q is > 4.95 %
SOR XIC B3:4/13 GRT R6:14.POS 0 GRT L13:59 L13:60 BST OTL B3:5/3 NXB ONS B3:2/9 ADD L13:157 1 L13:157 BND EOR
%   B3:4/13  "bypass" %
%   B3:5/3  TRACK5ERR %
%   L13:157  "I2 Avg queue over peak limit count" %
% Rung: 32 %
% average q is > rate-based limit %
SOR XIC B3:4/13 GRT R6:14.POS 0 GRT L13:59 L13:97 TON T4:15 0.001 150 0 EOR
%   B3:4/13  "bypass" %
%   L13:97  "i5 timed queue limit" %
% Rung: 33 %
% average q is > rate-based limit for 110 ms %
SOR XIC T4:15/EN XIC T4:15/DN BST OTL B3:5/3 NXB ONS B3:2/11 ADD L13:160 1 L13:160 BND EOR
%   B3:5/3  TRACK5ERR %
%   L13:160  "I2 Avg queue over timed limit count" %
% Rung: 34 %
SOR END EOR

LADDER 153 "INS5PASS"
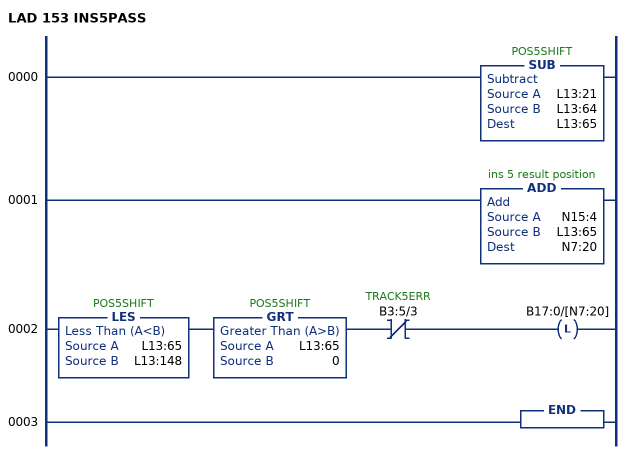
% Rung: 0 %
SOR SUB L13:21 L13:64 L13:65 EOR
%   L13:21  TOP_POSITION %
%   L13:64  POS5  "last acquisition position stamp" %
%   L13:65  POS5SHIFT %
% Rung: 1 %
SOR ADD N15:4 L13:65 N7:20 EOR
%   N15:4  INS_5_TRIG_LOC %
%   L13:65  POS5SHIFT %
%   N7:20  "ins 5 result position" %
% Rung: 2 %
SOR LES L13:65 L13:148 GRT L13:65 0 XIO B3:5/3 OTL B17:0/[N7:20] EOR
%   L13:65  POS5SHIFT %
%   L13:148  ALIGN_FAILS %
%   B3:5/3  TRACK5ERR %
%   N7:20  "ins 5 result position" %
% Rung: 3 %
SOR END EOR

LADDER 154 "INS5ACQ"
